FUNCTION F_UpdateEventTimeStamp
VAR_INPUT
	st_event : REFERENCE TO ST_Event;
END_VAR
VAR
	ulns: ULINT;
	fileTime: T_FILETIME;
END_VAR

ulns := F_GETSYSTEMTIME();
st_event.dtTimeStamp := F_SystemTimeToDT(nSystemTime:= ulns);

END_FUNCTION

(* stored: Version 1.1.0.1, ProductVersion 3.1.4024.12
   POU F_UpdateEventTimeStamp: Id {3e3e5dfe-3711-4edd-a58f-8af49b3b2532}, SpecialFunc None *)
